Universal Robots PolyScope program: Test_xmlrpc.urp

Program Test_xmlrpc (installation=default directory=/ursim/programs createdIn=5.21.3 lastSavedIn=5.21.3 robotSerialNumber=20195599999)
Calibrated DH parameters: a=[0, -0.425, -0.3922, 0, 0, 0]; d=[0.1625, 0, 0, 0.1333, 0.0997, 0.0996]; alpha=[1.570796, 0, 0, 1.570796, -1.570796, 0]; deltaTheta=[0, 0, 0, 0, 0, 0]
InitVariablesNode
BeforeStart
  Extend_pose := rpc_factory("xmlrpc","http://172.17.0.1:49211/RPC2")
Robot Program (runOnlyOnce=false)
  Current_pose := get_actual_tcp_pose()
  Recv_pose := Extend_pose.get_pose()
  Script: Current_pose[0]=Recv_pose.X
  Script: Current_pose[1]=Recv_pose.Y
  Script: Current_pose[2]=Recv_pose.Z
  Next_pose := Current_pose
  MoveJ speed 60 deg/s, acceleration 80 deg/s^2 (useActiveTCP=true optimoveEnabled=true optiMoveSpeed=0.3 optiMoveAcceleration=0.09) feature=Base
    Waypoint Variable (Variable): variable=Next_pose
